INTERFACE I_ChunkedRequestsMiddlewareConfig

METHOD PUBLIC TryGetHasMoreChunksFromRequest : BOOL
VAR_INPUT
	Request : I_Request;
	Destination : ANY;
END_VAR
END_METHOD

END_INTERFACE

(* stored: Version 1.1.0.1, ProductVersion 3.1.4024.12
   Itf I_ChunkedRequestsMiddlewareConfig: Id {693be1ca-178d-484a-aac4-a589765d99d8}
   Method TryGetHasMoreChunksFromRequest: Id {96dc9418-7dc1-4d0d-b401-8de66cb6107e} *)
